{attribute 'GeneratedUsingTerminal: AT2050-0500-0020'}
{attribute addProperty BoxType "AT2050-0500-0020"}
{attribute addProperty Id "A_0093_AT2020_5250_0019_AT2020_5250AT2020_01D6DEDF80"}
{attribute addProperty CRC "164429730"}
{attribute addProperty Size "80"}
TYPE A_0051_AT2050_0500_0020_09CCFFA2 EXTENDS AT2050_86175B41 :
STRUCT
	{attribute addProperty Name "A_0093_AT2020_5250_0019_AT2020_5250"}
	A_0093_AT2020_5250_0019_AT2020_5250 : AT2020_01D6DEDF;
END_STRUCT
END_TYPE

(* stored: Version 1.2.0.0, ProductVersion 3.1.4024.9
   DUT A_0051_AT2050_0500_0020_09CCFFA2: Id {f3dda276-58b4-4900-9214-e0c3026a9505} *)
